Fanuc KAREL source: compact_preamble.KL

PROGRAM KT00437
%NOLOCKGROUP
VAR
I1:INTEGER;I2:INTEGER;OUT:BOOLEAN
BEGIN
I1=2
I2=3
I1=2
I2=3
OUT=(I1 >=I2)
END KT00437
